FUNCTION_BLOCK LinkedListEnumerator EXTENDS EnumeratorBase IMPLEMENTS I_ForwardEnumerator
VAR
	linkedListFirstItem : REFERENCE TO I_LinkedListItem;
	currentItem : I_LinkedListItem;
	nextItem : I_LinkedListItem;
END_VAR

METHOD FB_init : BOOL
VAR_INPUT
	bInitRetains : BOOL; // if TRUE, the retain variables are initialized (warm start / cold start)
	bInCopyCode : BOOL;  // if TRUE, the instance afterwards gets moved into the copy code (online change)
	ConnectionUpdater : I_EnumeratorConnectionUpdater;
	LinkedListFirstItem : REFERENCE TO I_LinkedListItem;
END_VAR
THIS^.LinkedListFirstItem REF= LinkedListFirstItem;
END_METHOD

METHOD PUBLIC MoveNext : BOOL
VAR_INPUT
END_VAR
IF nextItem = 0 THEN
	currentItem := 0;
	RETURN;
END_IF

currentItem := nextItem;
nextItem := currentItem.Next;
END_METHOD

METHOD PROTECTED ABSTRACT OnGetValue : BOOL
VAR_INPUT
	Destination : ANY;
END_VAR
IF currentItem = 0 THEN
	RETURN;
END_IF

currentItem.Get(Destination);
END_METHOD

METHOD PROTECTED OnReset
VAR_INPUT
END_VAR
currentItem := 0;
nextItem := LinkedListFirstItem;
END_METHOD

END_FUNCTION_BLOCK

(* stored: Version 1.1.0.1, ProductVersion 3.1.4024.12
   POU LinkedListEnumerator: Id {c908c57f-ee22-4c86-a594-141eb5e0e7af}, SpecialFunc None
   Folder Constructor: Id {5ed93154-ab9d-468f-a6cc-f1798f080ae8}
   Folder Protected: Id {c2e0b2fd-7548-4204-89ed-8bd47fbf61f0}
   Method FB_init: Id {8c279887-c9ac-48ea-925e-99cb0ad2cec1}
   Method MoveNext: Id {e42b8db9-37db-4f9f-b8c0-718c5fcfec58}
   Method OnGetValue: Id {2131a1b1-137b-4505-ab83-f36e8ccf1f7d}
   Method OnReset: Id {ebef311d-589b-4c91-91bd-44321d33a333} *)
